# EPICS substitutions: iocs/MC05/MCApp/Db/SAI_8MotorStatus.substitutions
file /opt/epics/modules/SAI/db/SAI_8MotorStatus.db {
pattern {	ASYNPORT,	TMOT,		SCAN,		P,		R}
        { 	"pmac",		"1",		".2 second",	"XF:06BMA-OP","{Mir:M3}"}
	{ 	"pmac",		"1",		".2 second",	"XF:06BMA-BI","{Fltr:01}"}
}
